FUNCTION_BLOCK FB_TestChain1 EXTENDS FB_Chain
VAR_INPUT
END_VAR
VAR_OUTPUT
END_VAR
VAR
END_VAR

super^();

METHOD PROTECTED Busy : BOOL
VAR_INPUT
END_VAR
CASE fbStepWorkerBusy.uiStep OF

0:
	IF rChainController
		.releaseCheck(THIS^)
		.releaseFromChain(sChainReleasing := 'fbChain2', THIS^)
		.releaseResult(THIS^) 
	THEN
		fbStepWorkerInit.mNextStep(10);
	END_IF
10:
	;
20:
	;
30:

END_CASE
END_METHOD

METHOD PROTECTED Error : BOOL
VAR_INPUT
END_VAR
END_METHOD

METHOD PROTECTED Idle : BOOL
VAR_INPUT
END_VAR
END_METHOD

METHOD PROTECTED Init : BOOL
VAR_INPUT
END_VAR
Start();
END_METHOD

METHOD PROTECTED Prepare : BOOL
VAR_INPUT
END_VAR
END_METHOD

METHOD PROTECTED Ready : BOOL
VAR_INPUT
END_VAR
END_METHOD

METHOD PROTECTED Waiting : BOOL
VAR_INPUT
END_VAR
END_METHOD

END_FUNCTION_BLOCK

(* stored: Version 1.1.0.1, ProductVersion 3.1.4024.0
   POU FB_TestChain1: Id {743f7692-10f4-4273-a2c5-6e6083703b28}, SpecialFunc None
   Method Busy: Id {52999d6e-7318-424a-9025-f203b9d3dd83}
   Method Error: Id {ba9c29f6-dcc0-494d-ba38-a0a3f07552b0}
   Method Idle: Id {705993f9-2fe6-4427-bccd-0182dbc12a27}
   Method Init: Id {81bb4ced-ddc0-4275-a5e5-a2009b9dbcb0}
   Method Prepare: Id {5a64151a-9662-481a-9039-96016bcb6e31}
   Method Ready: Id {e7dcfe44-9fd7-4b37-8a66-909bcfe6c3f0}
   Method Waiting: Id {4ea2f4b0-0b9f-45e1-a68b-e8528cd295f3} *)
